SUBAPPLICATION AND_AUF (* Logisches UND (IN1 AND IN2) für AUF-Bedingung *)
  (* Standard: 61499-2 *)
  (* Version 1.0, 2025-01-15, franz, Meisterschulen am Ostbahnhof *)
  PACKAGE MyLib::sys;
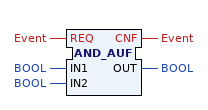
  EVENT_INPUT
    REQ;
  END_EVENT
  EVENT_OUTPUT
    CNF;
  END_EVENT
  VAR_INPUT
    IN1 : BOOL;
    IN2 : BOOL;
  END_VAR
  VAR_OUTPUT
    OUT : BOOL;
  END_VAR
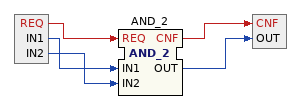
  FBS
    AND_2 : iec61131::bitwiseOperators::AND_2;
  END_FBS
  EVENT_CONNECTIONS
    REQ TO AND_2.REQ;
    AND_2.CNF TO CNF;
  END_CONNECTIONS
  DATA_CONNECTIONS
    IN1 TO AND_2.IN1;
    IN2 TO AND_2.IN2;
    AND_2.OUT TO OUT;
  END_CONNECTIONS
END_SUBAPPLICATION
